TYPE ST_Navigation_HMI :
STRUCT
	
END_STRUCT
END_TYPE

(* stored: Version 1.1.0.1
   DUT ST_Navigation_HMI: Id {73d5f465-8b78-4f4c-aead-5fffa3aace56} *)
